FUNCTION_BLOCK SafetyIO EXTENDS SM_SafetyIO
VAR_INPUT
END_VAR
VAR_OUTPUT
END_VAR
VAR
    _testVar : INT;
END_VAR

SUPER^();

// do stuff

//SUPER^();

END_FUNCTION_BLOCK

(* stored: Version 1.1.0.1, ProductVersion 3.1.4018.5
   POU SafetyIO: Id {d3ad2252-5181-4da1-86d8-740af3d7a27c}, SpecialFunc None *)
